FUNCTION_BLOCK PUBLISH_21 (* 6-Variable Publisher *)
  (* Standard: 61499-1; Classification: Communications *)
  (* Version 0.0, 2004-06-09, JHC, Rockwell Automation *)
  (* Compiler header: package fb.rt.net; *)
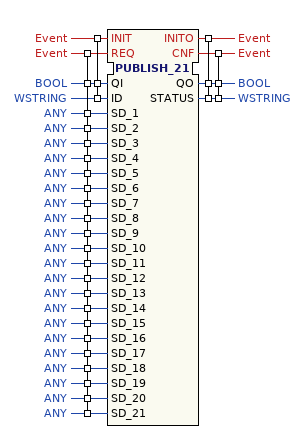
  EVENT_INPUT
    INIT WITH QI, ID; (* Service Initialization *)
    REQ WITH QI, SD_1, SD_2, SD_3, SD_4, SD_5, SD_6, SD_7, SD_8, SD_9, SD_10, SD_11, SD_12, SD_13, SD_14, SD_15, SD_16, SD_17, SD_18, SD_19, SD_20, SD_21; (* Service Request *)
  END_EVENT
  EVENT_OUTPUT
    INITO WITH QO, STATUS; (* Initialization Confirm *)
    CNF WITH QO, STATUS; (* Service Confirmation *)
  END_EVENT
  VAR_INPUT
    QI : BOOL; (* Event Input Qualifier *)
    ID : WSTRING; (* Connection Identifier *)
    SD_1 : ANY; (* Data to Send *)
    SD_2 : ANY; (* Data to Send *)
    SD_3 : ANY; (* Data to Send *)
    SD_4 : ANY; (* Data to Send *)
    SD_5 : ANY; (* Data to Send *)
    SD_6 : ANY; (* Data to Send *)
    SD_7 : ANY; (* Data to Send *)
    SD_8 : ANY; (* Data to Send *)
    SD_9 : ANY; (* Data to Send *)
    SD_10 : ANY; (* Data to Send *)
    SD_11 : ANY; (* Data to Send *)
    SD_12 : ANY; (* Data to Send *)
    SD_13 : ANY; (* Data to Send *)
    SD_14 : ANY; (* Data to Send *)
    SD_15 : ANY; (* Data to Send *)
    SD_16 : ANY; (* Data to Send *)
    SD_17 : ANY; (* Data to Send *)
    SD_18 : ANY; (* Data to Send *)
    SD_19 : ANY; (* Data to Send *)
    SD_20 : ANY; (* Data to Send *)
    SD_21 : ANY; (* Data to Send *)
  END_VAR
  VAR_OUTPUT
    QO : BOOL; (* Event Output Qualifier *)
    STATUS : WSTRING; (* Service Status *)
  END_VAR
END_FUNCTION_BLOCK
